FUNCTION QUARTERS_TO_DWORD
  (* Standard: 61499-1; Description: Copyright (c) 2024 HR Agrartechnik GmbH This program and the accompanying materials are made available under the terms of the Eclipse Public License 2.0 which is available at https://www.eclipse.org/legal/epl-2.0/ SPDX-License-Identifier: EPL-2.0 *)
  (* Version 1.0, 2024-02-22, franz *)
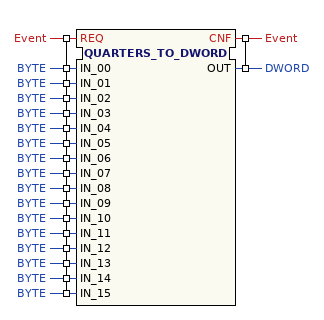
  EVENT_INPUT
    REQ WITH IN_00, IN_01, IN_02, IN_03, IN_04, IN_05, IN_06, IN_07, IN_08, IN_09, IN_10, IN_11, IN_12, IN_13, IN_14, IN_15; (* Normal Execution Request *)
  END_EVENT
  EVENT_OUTPUT
    CNF WITH OUT; (* Execution Confirmation *)
  END_EVENT
  VAR_INPUT
    IN_00 : BYTE; (* QUARTER BYTE 00 *)
    IN_01 : BYTE; (* QUARTER BYTE 01 *)
    IN_02 : BYTE; (* QUARTER BYTE 02 *)
    IN_03 : BYTE; (* QUARTER BYTE 03 *)
    IN_04 : BYTE; (* QUARTER BYTE 04 *)
    IN_05 : BYTE; (* QUARTER BYTE 05 *)
    IN_06 : BYTE; (* QUARTER BYTE 06 *)
    IN_07 : BYTE; (* QUARTER BYTE 07 *)
    IN_08 : BYTE; (* QUARTER BYTE 08 *)
    IN_09 : BYTE; (* QUARTER BYTE 09 *)
    IN_10 : BYTE; (* QUARTER BYTE 10 *)
    IN_11 : BYTE; (* QUARTER BYTE 11 *)
    IN_12 : BYTE; (* QUARTER BYTE 12 *)
    IN_13 : BYTE; (* QUARTER BYTE 13 *)
    IN_14 : BYTE; (* QUARTER BYTE 14 *)
    IN_15 : BYTE; (* QUARTER BYTE 15 *)
  END_VAR
  VAR_OUTPUT
    OUT : DWORD; (* DWORD Output *)
  END_VAR
  BODY IN ST:
FUNCTION QUARTERS_TO_DWORD

VAR_INPUT
	IN_00 : BYTE;    // QUARTER BYTE 00
	IN_01 : BYTE;    // QUARTER BYTE 01
	IN_02 : BYTE;    // QUARTER BYTE 02
	IN_03 : BYTE;    // QUARTER BYTE 03
	IN_04 : BYTE;    // QUARTER BYTE 04
	IN_05 : BYTE;    // QUARTER BYTE 05
	IN_06 : BYTE;    // QUARTER BYTE 06
	IN_07 : BYTE;    // QUARTER BYTE 07
	IN_08 : BYTE;    // QUARTER BYTE 08
	IN_09 : BYTE;    // QUARTER BYTE 09
	IN_10 : BYTE;    // QUARTER BYTE 10
	IN_11 : BYTE;    // QUARTER BYTE 11
	IN_12 : BYTE;    // QUARTER BYTE 12
	IN_13 : BYTE;    // QUARTER BYTE 13
	IN_14 : BYTE;    // QUARTER BYTE 14
	IN_15 : BYTE;    // QUARTER BYTE 15
END_VAR

VAR_OUTPUT
	OUT : DWORD;    // DWORD Output
END_VAR

(* this Function combines the 16 QUARTER BYTES to a dword *)
OUT := SHL(BYTE_TO_DWORD(IN_15), SHIFT_QUARTER_15)
	OR SHL(BYTE_TO_DWORD(IN_14), SHIFT_QUARTER_14)
	OR SHL(BYTE_TO_DWORD(IN_13), SHIFT_QUARTER_13)
	OR SHL(BYTE_TO_DWORD(IN_12), SHIFT_QUARTER_12)
	OR SHL(BYTE_TO_DWORD(IN_11), SHIFT_QUARTER_11)
	OR SHL(BYTE_TO_DWORD(IN_10), SHIFT_QUARTER_10)
	OR SHL(BYTE_TO_DWORD(IN_09), SHIFT_QUARTER_09)
	OR SHL(BYTE_TO_DWORD(IN_08), SHIFT_QUARTER_08)
	OR SHL(BYTE_TO_DWORD(IN_07), SHFT_QUARTER_07)
	OR SHL(BYTE_TO_DWORD(IN_06), SHFT_QUARTER_06)
	OR SHL(BYTE_TO_DWORD(IN_05), SHFT_QUARTER_05)
	OR SHL(BYTE_TO_DWORD(IN_04), SHFT_QUARTER_04)
	OR SHL(BYTE_TO_DWORD(IN_03), SHFT_QUARTER_03)
	OR SHL(BYTE_TO_DWORD(IN_02), SHFT_QUARTER_02)
	OR SHL(BYTE_TO_DWORD(IN_01), SHFT_QUARTER_01)
	OR SHL(BYTE_TO_DWORD(IN_00), SHFT_QUARTER_00);

END_FUNCTION
  END_BODY
END_FUNCTION
